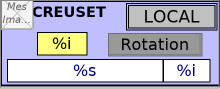
VISUALIZATION VISU_CREUSET_old  // 220x89
VAR_IN_OUT
	m_Input_CREUSET : BLOCK_IND_CR_379_TELEMARK;
END_VAR
    Rectangle (0,0 220x86)
    RoundedRectangle (37,32 50x23), "%i", text variable: m_Input_CREUSET.PRM_NCR, invisible if: NOT Global_Variables.PRG_USER.ACTU_USER.MAINTENANCE OR NOT MACHINE.State_manu
        OnMouseDown: write the text variable via InputWithLimits, min 1, max m_Input_CREUSET.CONF_NCR
    Rectangle (6,3 126x18), "CREUSET"
    RoundedRectangle (7,59 156x23), "%s", text variable: m_Input_CREUSET.STATE_MAT
    RoundedRectangle (163,59 47x23), "%i", text variable: m_Input_CREUSET.STATE_POS
    Button (108,33 94x23), "Rotation", invisible if: NOT m_Input_CREUSET.AUTOR_Change_IHM OR NOT PRG_User.ACTU_USER.MAINTENANCE
        tap m_Input_CREUSET.M_Change
    Image (1,-3 32x32), invisible if: NOT m_Input_CREUSET.State_nok, image: MesImages.warning
    RoundedRectangle (128,5 87x23), "REMOTE", invisible if: not m_Input_CREUSET.OUT_RMT
    RoundedRectangle (128,5 87x23), "LOCAL", invisible if: m_Input_CREUSET.OUT_RMT
    Rectangle (126,3 91x27), invisible if: Not m_Input_CREUSET.AUTOR_Remote_IHM, input disabled if: NOT PRG_User.ACTU_USER.MAINTENANCE
        tap m_Input_CREUSET.M_Remote
END_VISUALIZATION

(* stored: Version 1.1.0.1, ProductVersion 3.1.4026.18
   Visu VISU_CREUSET_old: Id {34569d39-0d9b-4b5b-b4e2-20c03314f7bf} *)
